// Mitsubishi GX Works2 project: PLC 적산 타이머   PLC: Q03UDV

PROGRAM MAIN
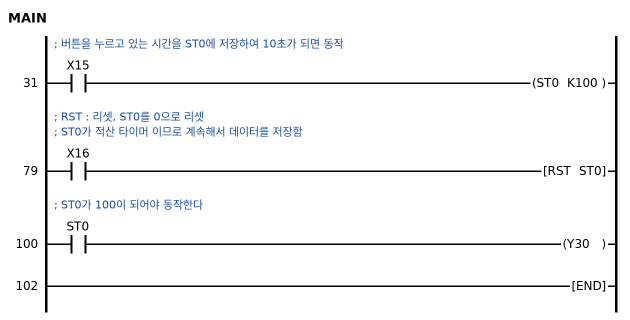
; 버튼을 누르고 있는 시간을 ST0에 저장하여 10초가 되면 동작
31    LD      X15
      OUT     ST0 K100
; RST : 리셋, ST0를 0으로 리셋
; ST0가 적산 타이머 이므로 계속해서 데이터를 저장함
79    LD      X16
      RST     ST0
; ST0가 100이 되어야 동작한다
100   LD      ST0
      OUT     Y30
102   END
END_PROGRAM
